// TIA Portal V17 export
// export: Created 2024-08-29T23:09:23.5181153Z, ExportSetting WithDefaults, DisplayName Totally Integrated Automation Portal, DisplayVersion V17 Update 7, DisplayName TIA Portal Openness, DisplayVersion V17 Update 7, DisplayName TIA Portal Version Control Interface, DisplayVersion V17, DisplayName SINAMICS Startdrive Advanced, DisplayVersion V17 SP2, DisplayName SINAMICS Startdrive G110M, G120, G120C, G120D, G120P, G115D, DisplayVersion V17 SP2, DisplayName SINAMICS Startdrive G130, G150, S120, S150, SINAMICS MV, S210, DisplayVersion V17 SP2, DisplayName STEP 7 Professional, DisplayVersion V17 Update 7, DisplayName STEP 7 Safety, DisplayVersion V17 Update 6, DisplayName WinCC Advanced / Unified PC, DisplayVersion V17 Update 7
FUNCTION "eksFC" : Void   // FC305, LAD
TITLE = Euchner Management EKS KEY
{ S7_Optimized_Access := 'FALSE' }
VERSION : 0.1
// stored: AutoNumber false, IsIECCheckEnabled false, SetENOAutomatically false, UDAEnableTagReadback false
   VAR_INPUT
      iKeyIn : Bool;
      iEksLevel : Byte;
      iEksEmployeeID : DWord;
      iEksKeyID1 : DWord;
      iEksKeyID2 : DWord;
      iEksJobFinished : Bool;
      hmiCurrentPage : Word;
   END_VAR
   VAR_OUTPUT
      qEksStartAdress : Byte;
      qEksDataLength : Byte;
      qEksData1 : Byte;
      qEksData2 : DWord;
      qEksWriteCommand : Bool;
   END_VAR
   VAR_TEMP
      tNone : Bool;
      tDBAddressKeys : Int;
      tDBAddressHMIPage : Int;
      tDBKeyStructLength : Int;
      tDBAddress : Int;
      tDBLength : Int;
      tCycle : Int;
      tFill : Int;
      tKey : "udt_EKS_KEY";
      tDBStartAddress : Int;
      tsearch : Bool;
      i : Int;
   END_VAR
   VAR CONSTANT
      DB : Byte := 16#84;
   END_VAR
   VAR_TEMP   // added for the SCL form of the ladder/FBD networks
      _w1 : Bool;
      _w2 : Bool;
   END_VAR
BEGIN

REGION Network 1: Initialize Temp Values
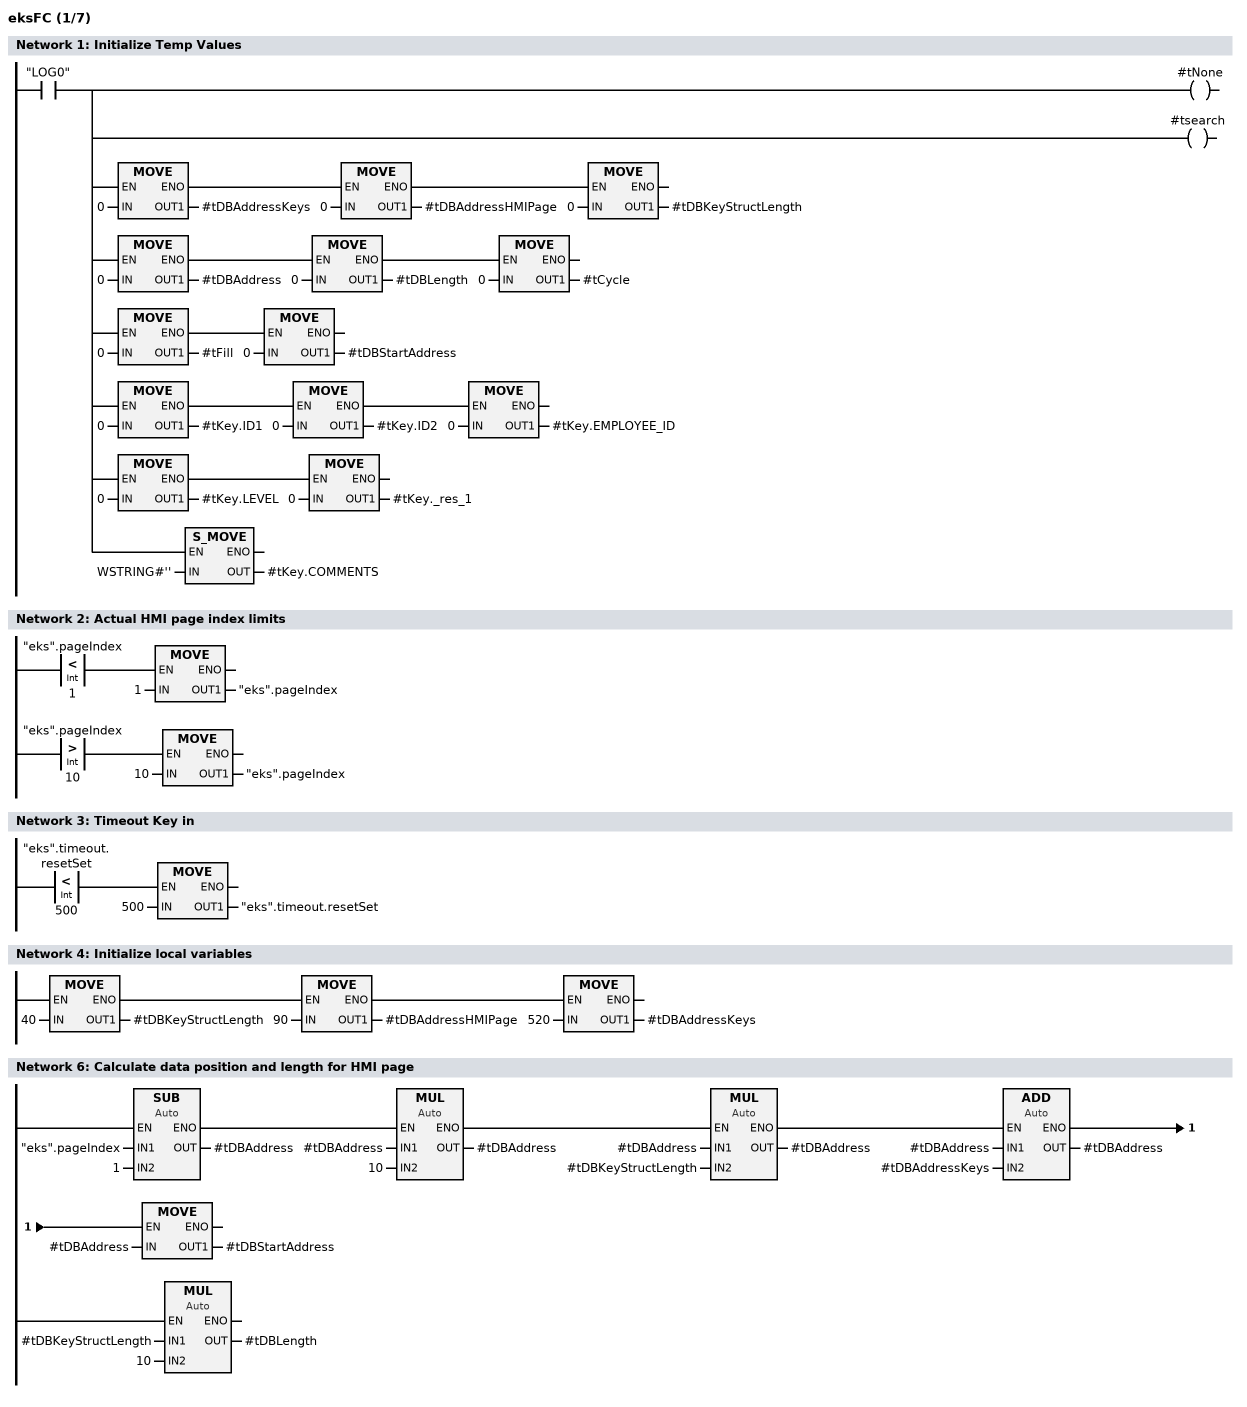
   RUNG wire#powerrail
      Contact( "LOG0" )
      wire#w1
      Coil( #tNone )
   END_RUNG
   RUNG wire#w1
      Coil( #tsearch )
   END_RUNG
   RUNG wire#w1
      Move(in := 0, out1 => #tDBAddressKeys)
      Move(in := 0, out1 => #tDBAddressHMIPage)
      Move(in := 0, out1 => #tDBKeyStructLength)
   END_RUNG
   RUNG wire#w1
      Move(in := 0, out1 => #tDBAddress)
      Move(in := 0, out1 => #tDBLength)
      Move(in := 0, out1 => #tCycle)
   END_RUNG
   RUNG wire#w1
      Move(in := 0, out1 => #tFill)
      Move(in := 0, out1 => #tDBStartAddress)
   END_RUNG
   RUNG wire#w1
      Move(in := 0, out1 => #tKey.ID1)
      Move(in := 0, out1 => #tKey.ID2)
      Move(in := 0, out1 => #tKey.EMPLOYEE_ID)
   END_RUNG
   RUNG wire#w1
      Move(in := 0, out1 => #tKey.LEVEL)
      Move(in := 0, out1 => #tKey._res_1)
   END_RUNG
   RUNG wire#w1
      S_Move(in := WSTRING#'', out => #tKey.COMMENTS)
   END_RUNG
   // the same network as SCL:
   #tNone := "LOG0";
   #tsearch := "LOG0";
   IF "LOG0" THEN
       #tDBAddressKeys := 0;
       #tDBAddressHMIPage := 0;
       #tDBKeyStructLength := 0;
       #tDBAddress := 0;
       #tDBLength := 0;
       #tCycle := 0;
       #tFill := 0;
       #tDBStartAddress := 0;
       #tKey.ID1 := 0;
       #tKey.ID2 := 0;
       #tKey.EMPLOYEE_ID := 0;
       #tKey.LEVEL := 0;
       #tKey._res_1 := 0;
       #tKey.COMMENTS := WSTRING#'';
   END_IF;
END_REGION

REGION Network 2: Actual HMI page index limits
   RUNG wire#powerrail
      { S7_Templates := "SrcType := Int" } LT_Contact(in1 := "eks".pageIndex, in2 := 1)
      Move(in := 1, out1 => "eks".pageIndex)
   END_RUNG
   RUNG wire#powerrail
      { S7_Templates := "SrcType := Int" } GT_Contact(in1 := "eks".pageIndex, in2 := 10)
      Move(in := 10, out1 => "eks".pageIndex)
   END_RUNG
   // the same network as SCL:
   IF "eks".pageIndex < 1 THEN "eks".pageIndex := 1; END_IF;
   IF "eks".pageIndex > 10 THEN "eks".pageIndex := 10; END_IF;
END_REGION

REGION Network 3: Timeout Key in
   RUNG wire#powerrail
      { S7_Templates := "SrcType := Int" } LT_Contact(in1 := "eks".timeout.resetSet, in2 := 500)
      Move(in := 500, out1 => "eks".timeout.resetSet)
   END_RUNG
   // the same network as SCL:
   IF "eks".timeout.resetSet < 500 THEN "eks".timeout.resetSet := 500; END_IF;
END_REGION

REGION Network 4: Initialize local variables
   RUNG wire#powerrail
      Move(in := 40, out1 => #tDBKeyStructLength)
      Move(in := 90, out1 => #tDBAddressHMIPage)
      Move(in := 520, out1 => #tDBAddressKeys)
   END_RUNG
   // the same network as SCL:
   #tDBKeyStructLength := 40;
   #tDBAddressHMIPage := 90;
   #tDBAddressKeys := 520;
END_REGION

REGION Network 6: Calculate data position and length for HMI page
   RUNG wire#powerrail
      Sub(in1 := "eks".pageIndex, in2 := 1, out => #tDBAddress)
      Mul(in1 := #tDBAddress, in2 := 10, out => #tDBAddress)
      Mul(in1 := #tDBAddress, in2 := #tDBKeyStructLength, out => #tDBAddress)
      Add(in1 := #tDBAddress, in2 := #tDBAddressKeys, out => #tDBAddress)
      Move(in := #tDBAddress, out1 => #tDBStartAddress)
   END_RUNG
   RUNG wire#powerrail
      Mul(in1 := #tDBKeyStructLength, in2 := 10, out => #tDBLength)
   END_RUNG
   // the same network as SCL:
   #tDBAddress := "eks".pageIndex - 1;
   #tDBAddress := #tDBAddress * 10;
   #tDBAddress := #tDBAddress * #tDBKeyStructLength;
   #tDBAddress := #tDBAddress + #tDBAddressKeys;
   #tDBStartAddress := #tDBAddress;
   #tDBLength := #tDBKeyStructLength * 10;
END_REGION

REGION Network 7 (SCL): Copy data for page (10 keys)
   POKE_BLK(area_src:=#DB,
            dbNumber_src:=305,
            byteOffset_src:=#tDBAddress,
            area_dest:=#DB,
            dbNumber_dest:=305,
            byteOffset_dest:=90,
            count:=#tDBLength);
END_REGION

REGION Network 9: Inserted key
   // Store_Key_In is used to display only 1 time the level of euchner during storage function.
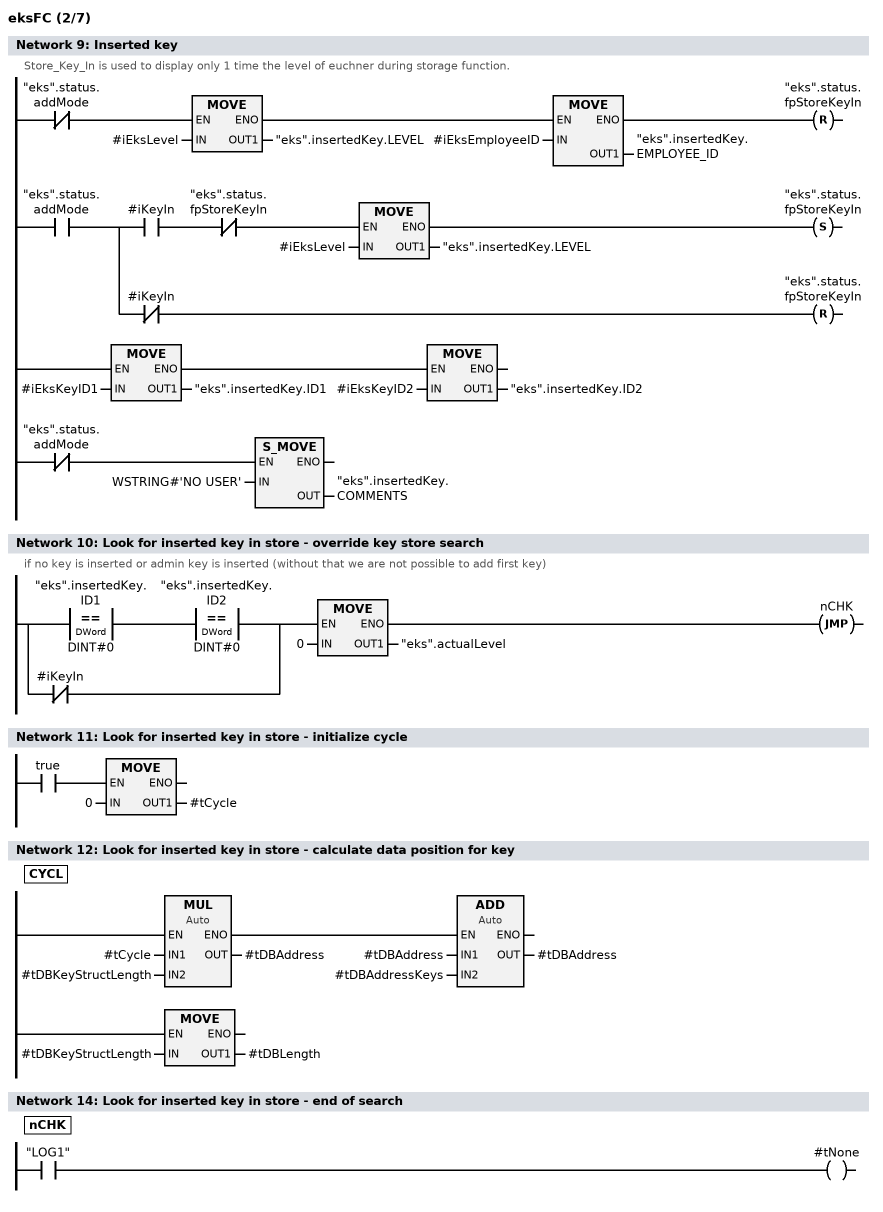
   RUNG wire#powerrail
      I_Contact( "eks".status.addMode )
      Move(in := #iEksLevel, out1 => "eks".insertedKey.LEVEL)
      Move(in := #iEksEmployeeID, out1 => "eks".insertedKey.EMPLOYEE_ID)
      R_Coil( "eks".status.fpStoreKeyIn )
   END_RUNG
   RUNG wire#powerrail
      Contact( "eks".status.addMode )
      wire#w1
      Contact( #iKeyIn )
      I_Contact( "eks".status.fpStoreKeyIn )
      Move(in := #iEksLevel, out1 => "eks".insertedKey.LEVEL)
      S_Coil( "eks".status.fpStoreKeyIn )
   END_RUNG
   RUNG wire#w1
      I_Contact( #iKeyIn )
      R_Coil( "eks".status.fpStoreKeyIn )
   END_RUNG
   RUNG wire#powerrail
      Move(in := #iEksKeyID1, out1 => "eks".insertedKey.ID1)
      Move(in := #iEksKeyID2, out1 => "eks".insertedKey.ID2)
   END_RUNG
   RUNG wire#powerrail
      I_Contact( "eks".status.addMode )
      S_Move(in := WSTRING#'NO USER', out => "eks".insertedKey.COMMENTS)
   END_RUNG
   // the same network as SCL:
   IF NOT "eks".status.addMode THEN
       "eks".insertedKey.LEVEL := #iEksLevel;
       "eks".insertedKey.EMPLOYEE_ID := #iEksEmployeeID;
       "eks".status.fpStoreKeyIn := FALSE;
   END_IF;
   IF "eks".status.addMode AND #iKeyIn AND NOT "eks".status.fpStoreKeyIn THEN
       "eks".insertedKey.LEVEL := #iEksLevel;
       "eks".status.fpStoreKeyIn := TRUE;
   END_IF;
   IF "eks".status.addMode AND NOT #iKeyIn THEN "eks".status.fpStoreKeyIn := FALSE; END_IF;
   "eks".insertedKey.ID1 := #iEksKeyID1;
   "eks".insertedKey.ID2 := #iEksKeyID2;
   IF NOT "eks".status.addMode THEN "eks".insertedKey.COMMENTS := WSTRING#'NO USER'; END_IF;
END_REGION

REGION Network 10: Look for inserted key in store - override key store search
   // if no key is inserted or admin key is inserted (without that we are not possible to add first key)
   RUNG wire#powerrail
      { S7_Templates := "SrcType := DWord" } EQ_Contact(in1 := "eks".insertedKey.ID1, in2 := DINT#0)
      { S7_Templates := "SrcType := DWord" } EQ_Contact(in1 := "eks".insertedKey.ID2, in2 := DINT#0)
      wire#w1
      Move(in := 0, out1 => "eks".actualLevel)
      JumpCoil( nCHK )
   END_RUNG
   RUNG wire#powerrail
      I_Contact( #iKeyIn )
   END_RUNG wire#w1
   // the same network as SCL:
   #_w1 := (("eks".insertedKey.ID1 = DINT#0) AND ("eks".insertedKey.ID2 = DINT#0)) OR NOT #iKeyIn;
   IF #_w1 THEN
       "eks".actualLevel := 0;
       GOTO nCHK;
   END_IF;
END_REGION

REGION Network 11: Look for inserted key in store - initialize cycle
   RUNG wire#powerrail
      Contact( true )
      Move(in := 0, out1 => #tCycle)
   END_RUNG
   // the same network as SCL:
   IF true THEN #tCycle := 0; END_IF;
END_REGION

REGION Network 12: Look for inserted key in store - calculate data position for key
   Label( CYCL )
   RUNG wire#powerrail
      Mul(in1 := #tCycle, in2 := #tDBKeyStructLength, out => #tDBAddress)
      Add(in1 := #tDBAddress, in2 := #tDBAddressKeys, out => #tDBAddress)
   END_RUNG
   RUNG wire#powerrail
      Move(in := #tDBKeyStructLength, out1 => #tDBLength)
   END_RUNG
   // the same network as SCL:
   CYCL:
   #tDBAddress := #tCycle * #tDBKeyStructLength;
   #tDBAddress := #tDBAddress + #tDBAddressKeys;
   #tDBLength := #tDBKeyStructLength;
END_REGION

REGION Network 13 (SCL): Look for inserted key in store - check ID of stored key
   FOR #i := 1 TO 130 DO
       #tKey := "eks".keys[#i];
       IF (#tKey.ID1 = "eks".insertedKey.ID1) AND
           (#tKey.ID2 = "eks".insertedKey.ID2) THEN
           "eks".actualLevel := #tKey.LEVEL;
           "eks".insertedKey.COMMENTS := #tKey.COMMENTS;
           EXIT;
       END_IF;
   END_FOR;
END_REGION

REGION Network 14: Look for inserted key in store - end of search
   Label( nCHK )
   RUNG wire#powerrail
      Contact( "LOG1" )
      Coil( #tNone )
   END_RUNG
   // the same network as SCL:
   nCHK:
   #tNone := "LOG1";
END_REGION

REGION Network 15: Reset of EKS higher levels until key is removed
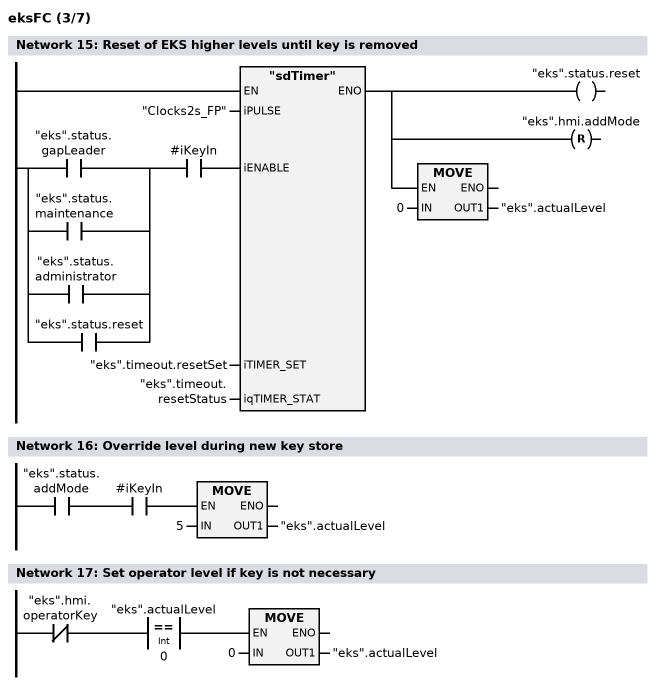
   RUNG wire#powerrail
      "sdTimer"(iENABLE := wire#w2, iPULSE := "Clocks2s_FP", iTIMER_SET := "eks".timeout.resetSet, iqTIMER_STAT := "eks".timeout.resetStatus)
      wire#w3
      Coil( "eks".status.reset )
   END_RUNG
   RUNG wire#powerrail
      Contact( "eks".status.gapLeader )
      wire#w1
      Contact( #iKeyIn )
   END_RUNG wire#w2
   RUNG wire#powerrail
      Contact( "eks".status.maintenance )
   END_RUNG wire#w1
   RUNG wire#powerrail
      Contact( "eks".status.administrator )
   END_RUNG wire#w1
   RUNG wire#powerrail
      Contact( "eks".status.reset )
   END_RUNG wire#w1
   RUNG wire#w3
      R_Coil( "eks".hmi.addMode )
   END_RUNG
   RUNG wire#w3
      Move(in := 0, out1 => "eks".actualLevel)
   END_RUNG
   // the same network as SCL:
   "sdTimer"(iPULSE := "Clocks2s_FP",
             iENABLE := ("eks".status.gapLeader OR "eks".status.maintenance OR "eks".status.administrator OR "eks".status.reset) AND #iKeyIn,
             iTIMER_SET := "eks".timeout.resetSet,
             iqTIMER_STAT := "eks".timeout.resetStatus,
             ENO => #_w1);
   "eks".status.reset := #_w1;
   IF #_w1 THEN
       "eks".hmi.addMode := FALSE;
       "eks".actualLevel := 0;
   END_IF;
END_REGION

REGION Network 16: Override level during new key store
   RUNG wire#powerrail
      Contact( "eks".status.addMode )
      Contact( #iKeyIn )
      Move(in := 5, out1 => "eks".actualLevel)
   END_RUNG
   // the same network as SCL:
   IF "eks".status.addMode AND #iKeyIn THEN "eks".actualLevel := 5; END_IF;
END_REGION

REGION Network 17: Set operator level if key is not necessary
   RUNG wire#powerrail
      I_Contact( "eks".hmi.operatorKey )
      { S7_Templates := "SrcType := Int" } EQ_Contact(in1 := "eks".actualLevel, in2 := 0)
      Move(in := 0, out1 => "eks".actualLevel)
   END_RUNG
   // the same network as SCL:
   IF NOT "eks".hmi.operatorKey AND ("eks".actualLevel = 0) THEN "eks".actualLevel := 0; END_IF;
END_REGION

REGION Network 18: EKS levels
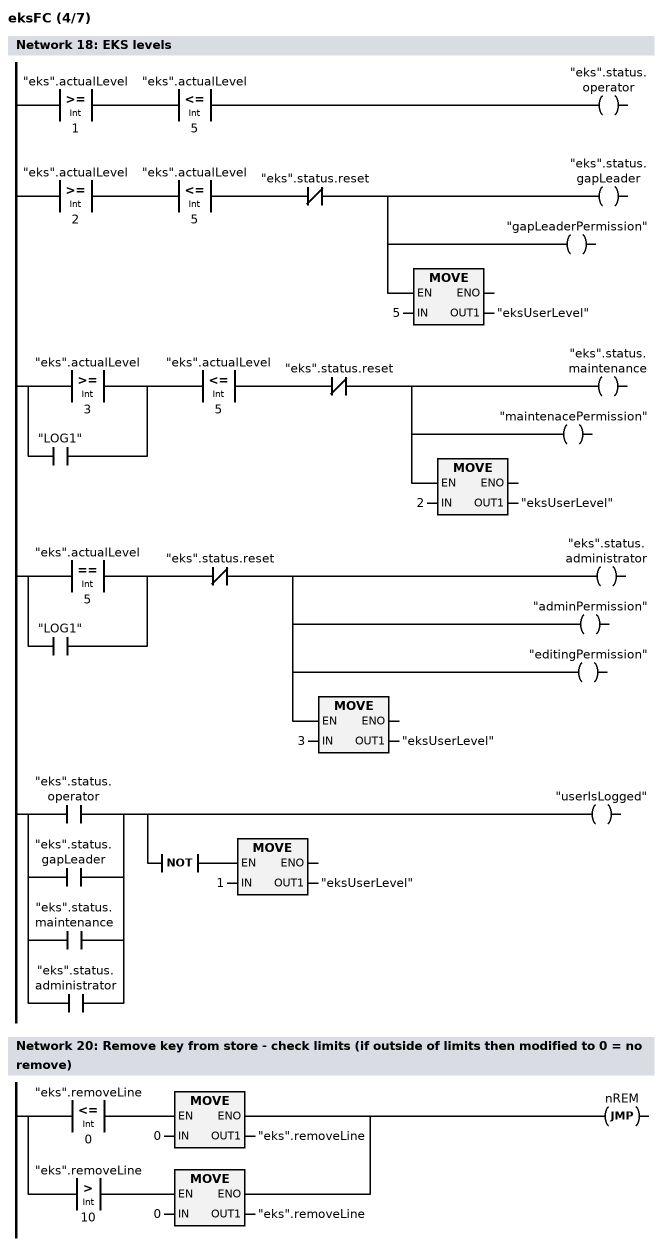
   RUNG wire#powerrail
      { S7_Templates := "SrcType := Int" } GE_Contact(in1 := "eks".actualLevel, in2 := 1)
      { S7_Templates := "SrcType := Int" } LE_Contact(in1 := "eks".actualLevel, in2 := 5)
      Coil( "eks".status.operator )
   END_RUNG
   RUNG wire#powerrail
      { S7_Templates := "SrcType := Int" } GE_Contact(in1 := "eks".actualLevel, in2 := 2)
      { S7_Templates := "SrcType := Int" } LE_Contact(in1 := "eks".actualLevel, in2 := 5)
      I_Contact( "eks".status.reset )
      wire#w1
      Coil( "eks".status.gapLeader )
   END_RUNG
   RUNG wire#w1
      Coil( "gapLeaderPermission" )
   END_RUNG
   RUNG wire#w1
      Move(in := 5, out1 => "eksUserLevel")
   END_RUNG
   RUNG wire#powerrail
      { S7_Templates := "SrcType := Int" } GE_Contact(in1 := "eks".actualLevel, in2 := 3)
      wire#w2
      { S7_Templates := "SrcType := Int" } LE_Contact(in1 := "eks".actualLevel, in2 := 5)
      I_Contact( "eks".status.reset )
      wire#w3
      Coil( "eks".status.maintenance )
   END_RUNG
   RUNG wire#powerrail
      Contact( "LOG1" )
   END_RUNG wire#w2
   RUNG wire#w3
      Coil( "maintenacePermission" )
   END_RUNG
   RUNG wire#w3
      Move(in := 2, out1 => "eksUserLevel")
   END_RUNG
   RUNG wire#powerrail
      { S7_Templates := "SrcType := Int" } EQ_Contact(in1 := "eks".actualLevel, in2 := 5)
      wire#w4
      I_Contact( "eks".status.reset )
      wire#w5
      Coil( "eks".status.administrator )
   END_RUNG
   RUNG wire#powerrail
      Contact( "LOG1" )
   END_RUNG wire#w4
   RUNG wire#w5
      Coil( "adminPermission" )
   END_RUNG
   RUNG wire#w5
      Coil( "editingPermission" )
   END_RUNG
   RUNG wire#w5
      Move(in := 3, out1 => "eksUserLevel")
   END_RUNG
   RUNG wire#powerrail
      Contact( "eks".status.operator )
      wire#w6
      Coil( "userIsLogged" )
   END_RUNG
   RUNG wire#powerrail
      Contact( "eks".status.gapLeader )
   END_RUNG wire#w6
   RUNG wire#powerrail
      Contact( "eks".status.maintenance )
   END_RUNG wire#w6
   RUNG wire#powerrail
      Contact( "eks".status.administrator )
   END_RUNG wire#w6
   RUNG wire#w6
      Not()
      Move(in := 1, out1 => "eksUserLevel")
   END_RUNG
   // the same network as SCL:
   "eks".status.operator := ("eks".actualLevel >= 1) AND ("eks".actualLevel <= 5);
   "eks".status.gapLeader := ("eks".actualLevel >= 2) AND ("eks".actualLevel <= 5) AND NOT "eks".status.reset;
   "gapLeaderPermission" := "eks".status.gapLeader;
   IF "eks".status.gapLeader THEN "eksUserLevel" := 5; END_IF;
   "eks".status.maintenance := (("eks".actualLevel >= 3) OR "LOG1") AND ("eks".actualLevel <= 5) AND NOT "eks".status.reset;
   "maintenacePermission" := "eks".status.maintenance;
   IF "eks".status.maintenance THEN "eksUserLevel" := 2; END_IF;
   "eks".status.administrator := (("eks".actualLevel = 5) OR "LOG1") AND NOT "eks".status.reset;
   "adminPermission" := "eks".status.administrator;
   "editingPermission" := "eks".status.administrator;
   IF "eks".status.administrator THEN "eksUserLevel" := 3; END_IF;
   "userIsLogged" := "eks".status.operator OR "eks".status.gapLeader OR "eks".status.maintenance OR "eks".status.administrator;
   IF NOT "userIsLogged" THEN "eksUserLevel" := 1; END_IF;
END_REGION

REGION Network 20: Remove key from store - check limits (if outside of limits then modified to 0 = no remove)
   RUNG wire#powerrail
      { S7_Templates := "SrcType := Int" } LE_Contact(in1 := "eks".removeLine, in2 := 0)
      Move(in := 0, out1 => "eks".removeLine)
      wire#w1
      JumpCoil( nREM )
   END_RUNG
   RUNG wire#powerrail
      { S7_Templates := "SrcType := Int" } GT_Contact(in1 := "eks".removeLine, in2 := 10)
      Move(in := 0, out1 => "eks".removeLine)
   END_RUNG wire#w1
   // the same network as SCL:
   #_w1 := "eks".removeLine <= 0;
   IF #_w1 THEN "eks".removeLine := 0; END_IF;
   #_w2 := "eks".removeLine > 10;
   IF #_w2 THEN "eks".removeLine := 0; END_IF;
   IF #_w1 OR #_w2 THEN GOTO nREM; END_IF;
END_REGION

REGION Network 21: Remove key from store - calculate data position and length for HMI page
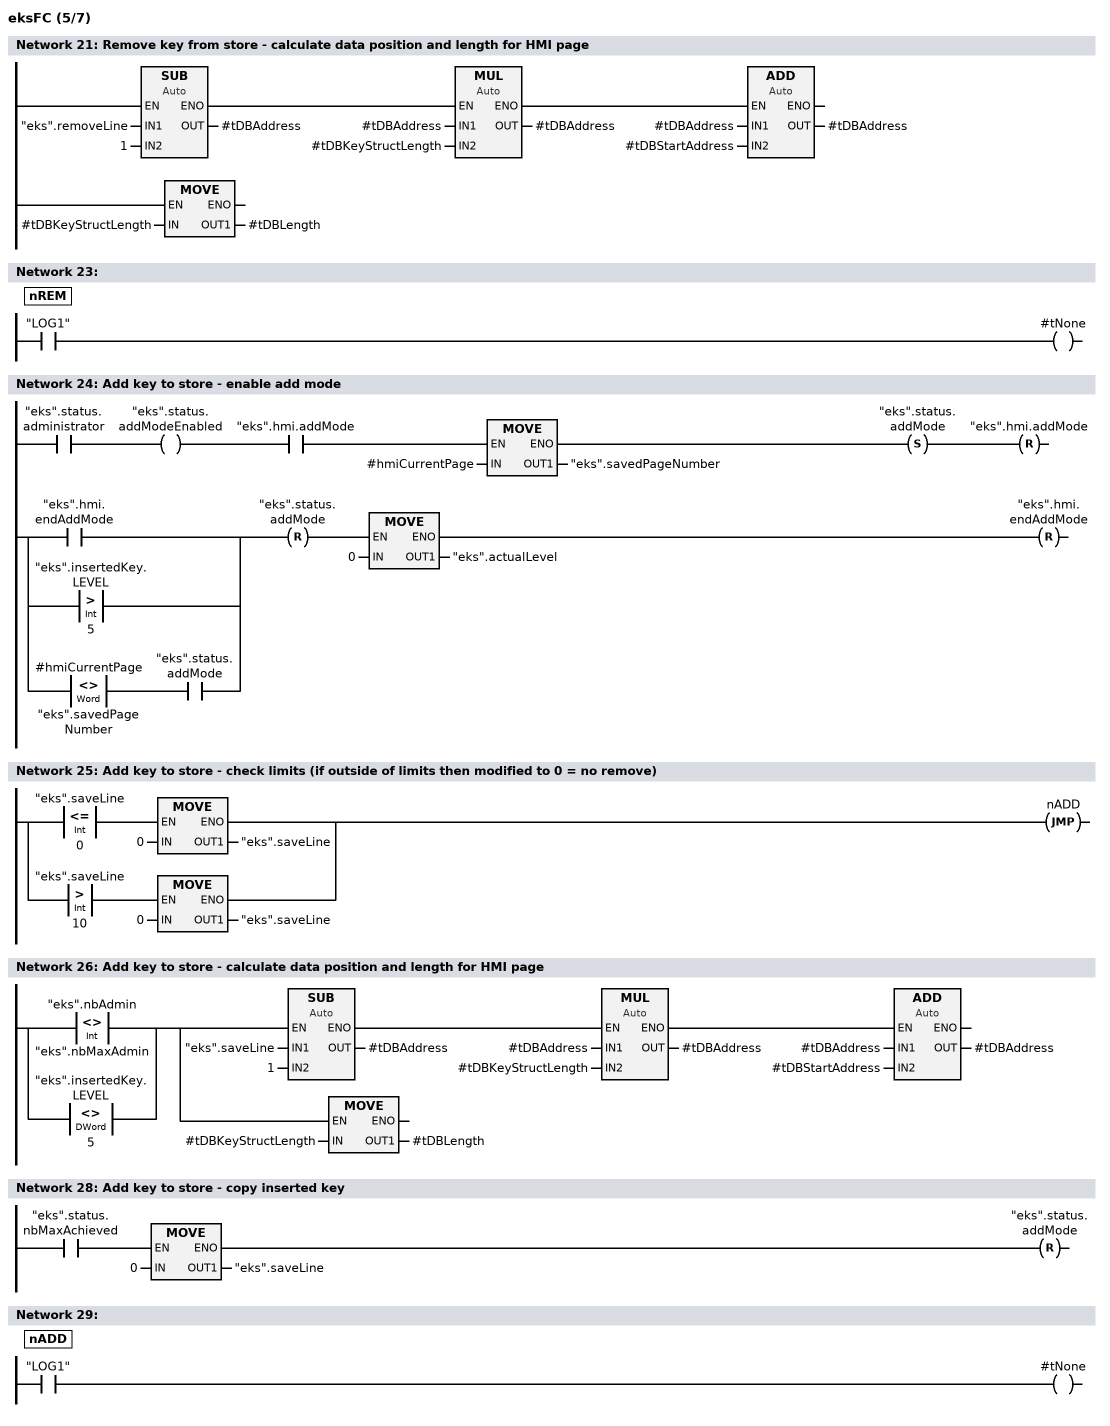
   RUNG wire#powerrail
      Sub(in1 := "eks".removeLine, in2 := 1, out => #tDBAddress)
      Mul(in1 := #tDBAddress, in2 := #tDBKeyStructLength, out => #tDBAddress)
      Add(in1 := #tDBAddress, in2 := #tDBStartAddress, out => #tDBAddress)
   END_RUNG
   RUNG wire#powerrail
      Move(in := #tDBKeyStructLength, out1 => #tDBLength)
   END_RUNG
   // the same network as SCL:
   #tDBAddress := "eks".removeLine - 1;
   #tDBAddress := #tDBAddress * #tDBKeyStructLength;
   #tDBAddress := #tDBAddress + #tDBStartAddress;
   #tDBLength := #tDBKeyStructLength;
END_REGION

REGION Network 22 (SCL): Remove key from store - delete key
   #tFill := 0;

   POKE_BLK(area_src:=#DB,
            dbNumber_src:=305,
            byteOffset_src:=5720,
            area_dest:=#DB,
            dbNumber_dest:=305,
            byteOffset_dest:=#tDBAddress,
            count:=#tDBLength);

   "eks".removeLine := 0;
END_REGION

REGION Network 23
   Label( nREM )
   RUNG wire#powerrail
      Contact( "LOG1" )
      Coil( #tNone )
   END_RUNG
   // the same network as SCL:
   nREM:
   #tNone := "LOG1";
END_REGION

REGION Network 24: Add key to store - enable add mode
   RUNG wire#powerrail
      Contact( "eks".status.administrator )
      Coil( "eks".status.addModeEnabled )
      Contact( "eks".hmi.addMode )
      Move(in := #hmiCurrentPage, out1 => "eks".savedPageNumber)
      S_Coil( "eks".status.addMode )
      R_Coil( "eks".hmi.addMode )
   END_RUNG
   RUNG wire#powerrail
      Contact( "eks".hmi.endAddMode )
      wire#w1
      R_Coil( "eks".status.addMode )
      Move(in := 0, out1 => "eks".actualLevel)
      R_Coil( "eks".hmi.endAddMode )
   END_RUNG
   RUNG wire#powerrail
      { S7_Templates := "SrcType := Int" } GT_Contact(in1 := "eks".insertedKey.LEVEL, in2 := 5)
   END_RUNG wire#w1
   RUNG wire#powerrail
      { S7_Templates := "SrcType := Word" } NE_Contact(in1 := #hmiCurrentPage, in2 := "eks".savedPageNumber)
      Contact( "eks".status.addMode )
   END_RUNG wire#w1
   // the same network as SCL:
   "eks".status.addModeEnabled := "eks".status.administrator;
   IF "eks".status.administrator AND "eks".hmi.addMode THEN
       "eks".savedPageNumber := #hmiCurrentPage;
       "eks".status.addMode := TRUE;
       "eks".hmi.addMode := FALSE;
   END_IF;
   #_w1 := "eks".hmi.endAddMode OR ("eks".insertedKey.LEVEL > 5) OR ((#hmiCurrentPage <> "eks".savedPageNumber) AND "eks".status.addMode);
   IF #_w1 THEN
       "eks".status.addMode := FALSE;
       "eks".actualLevel := 0;
       "eks".hmi.endAddMode := FALSE;
   END_IF;
END_REGION

REGION Network 25: Add key to store - check limits (if outside of limits then modified to 0 = no remove)
   RUNG wire#powerrail
      { S7_Templates := "SrcType := Int" } LE_Contact(in1 := "eks".saveLine, in2 := 0)
      Move(in := 0, out1 => "eks".saveLine)
      wire#w1
      JumpCoil( nADD )
   END_RUNG
   RUNG wire#powerrail
      { S7_Templates := "SrcType := Int" } GT_Contact(in1 := "eks".saveLine, in2 := 10)
      Move(in := 0, out1 => "eks".saveLine)
   END_RUNG wire#w1
   // the same network as SCL:
   #_w1 := "eks".saveLine <= 0;
   IF #_w1 THEN "eks".saveLine := 0; END_IF;
   #_w2 := "eks".saveLine > 10;
   IF #_w2 THEN "eks".saveLine := 0; END_IF;
   IF #_w1 OR #_w2 THEN GOTO nADD; END_IF;
END_REGION

REGION Network 26: Add key to store - calculate data position and length for HMI page
   RUNG wire#powerrail
      { S7_Templates := "SrcType := Int" } NE_Contact(in1 := "eks".nbAdmin, in2 := "eks".nbMaxAdmin)
      wire#w1
      Sub(in1 := "eks".saveLine, in2 := 1, out => #tDBAddress)
      Mul(in1 := #tDBAddress, in2 := #tDBKeyStructLength, out => #tDBAddress)
      Add(in1 := #tDBAddress, in2 := #tDBStartAddress, out => #tDBAddress)
   END_RUNG
   RUNG wire#powerrail
      { S7_Templates := "SrcType := DWord" } NE_Contact(in1 := "eks".insertedKey.LEVEL, in2 := 5)
   END_RUNG wire#w1
   RUNG wire#w1
      Move(in := #tDBKeyStructLength, out1 => #tDBLength)
   END_RUNG
   // the same network as SCL:
   IF ("eks".nbAdmin <> "eks".nbMaxAdmin) OR ("eks".insertedKey.LEVEL <> 5) THEN
       #tDBAddress := "eks".saveLine - 1;
       #tDBAddress := #tDBAddress * #tDBKeyStructLength;
       #tDBAddress := #tDBAddress + #tDBStartAddress;
       #tDBLength := #tDBKeyStructLength;
   END_IF;
END_REGION

REGION Network 27 (SCL): Add key to store - copy inserted key
   IF ("eks".insertedKey.LEVEL = 5  & NOT "eks".status.nbMaxAchieved) OR
       ("eks".insertedKey.LEVEL <> 5) THEN
       POKE_BLK(area_src := #DB,
                dbNumber_src := 305,
                byteOffset_src := 50,
                area_dest := #DB,
                dbNumber_dest := 305,
                byteOffset_dest := #tDBAddress,
                count := #tDBLength);
      "eks".saveLine := 0;
   END_IF;
END_REGION

REGION Network 28: Add key to store - copy inserted key
   RUNG wire#powerrail
      Contact( "eks".status.nbMaxAchieved )
      Move(in := 0, out1 => "eks".saveLine)
      R_Coil( "eks".status.addMode )
   END_RUNG
   // the same network as SCL:
   IF "eks".status.nbMaxAchieved THEN
       "eks".saveLine := 0;
       "eks".status.addMode := FALSE;
   END_IF;
END_REGION

REGION Network 29
   Label( nADD )
   RUNG wire#powerrail
      Contact( "LOG1" )
      Coil( #tNone )
   END_RUNG
   // the same network as SCL:
   nADD:
   #tNone := "LOG1";
END_REGION

REGION Network 30
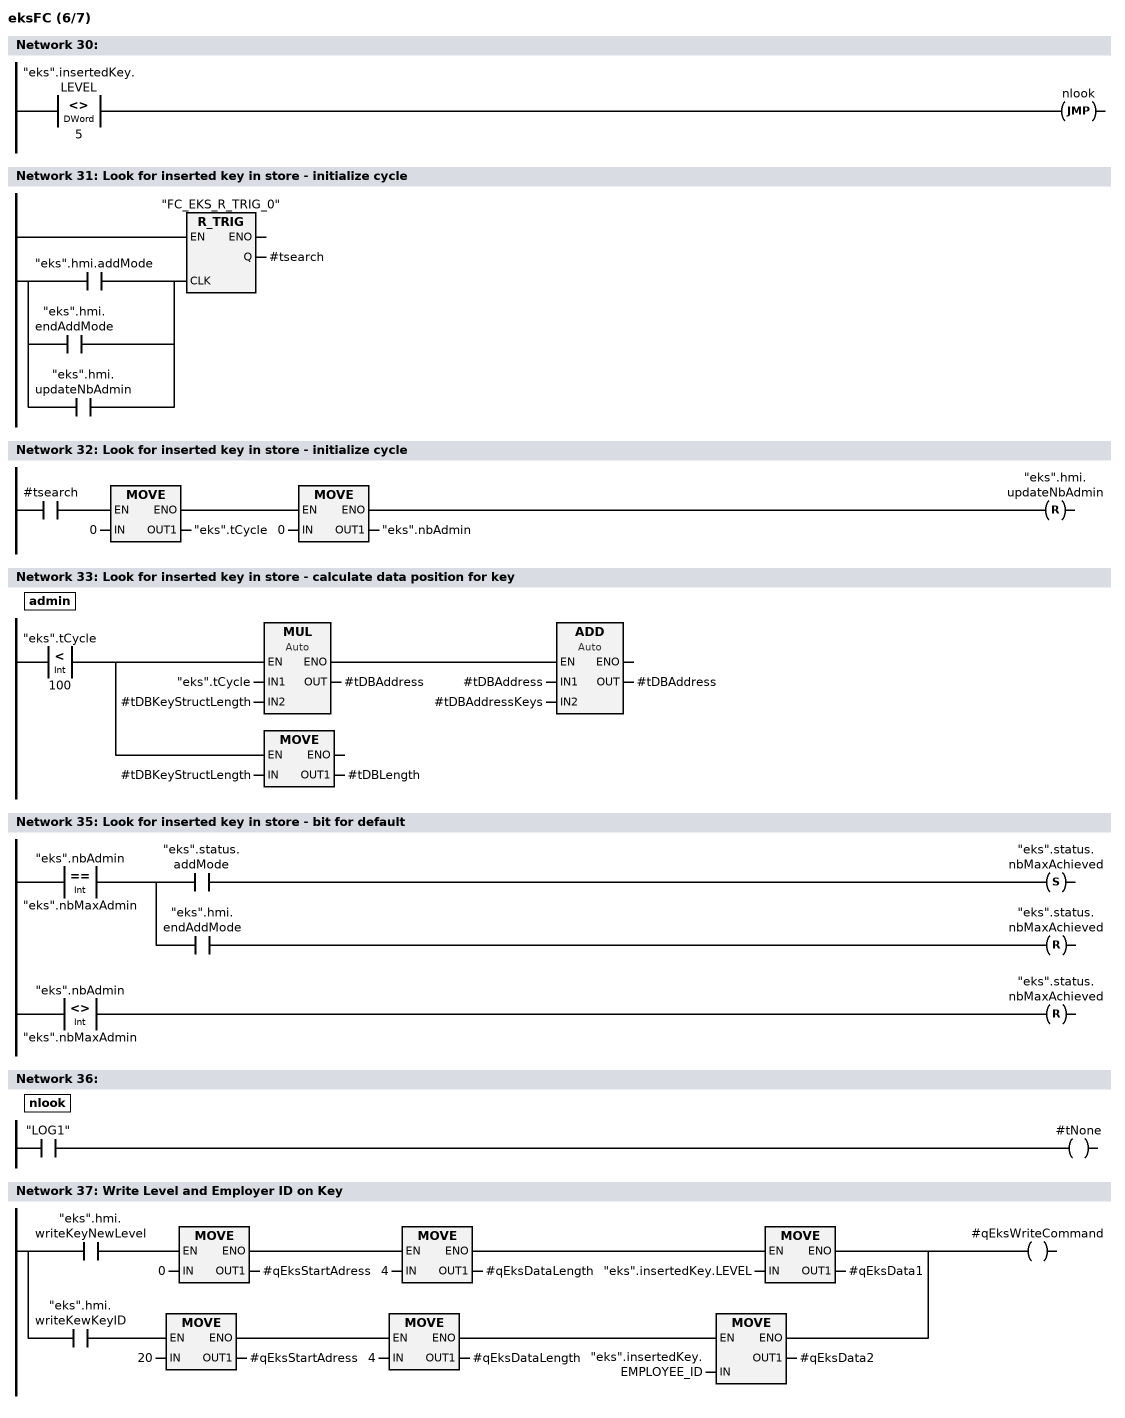
   RUNG wire#powerrail
      { S7_Templates := "SrcType := DWord" } NE_Contact(in1 := "eks".insertedKey.LEVEL, in2 := 5)
      JumpCoil( nlook )
   END_RUNG
   // the same network as SCL:
   IF "eks".insertedKey.LEVEL <> 5 THEN GOTO nlook; END_IF;
END_REGION

REGION Network 31: Look for inserted key in store - initialize cycle
   RUNG wire#powerrail
      "FC_EKS_R_TRIG_0".R_TRIG(CLK := wire#w1, Q => #tsearch)
   END_RUNG
   RUNG wire#powerrail
      Contact( "eks".hmi.addMode )
   END_RUNG wire#w1
   RUNG wire#powerrail
      Contact( "eks".hmi.endAddMode )
   END_RUNG wire#w1
   RUNG wire#powerrail
      Contact( "eks".hmi.updateNbAdmin )
   END_RUNG wire#w1
   // the same network as SCL:
   "FC_EKS_R_TRIG_0"(CLK := "eks".hmi.addMode OR "eks".hmi.endAddMode OR "eks".hmi.updateNbAdmin, Q => #tsearch);   // R_TRIG
END_REGION

REGION Network 32: Look for inserted key in store - initialize cycle
   RUNG wire#powerrail
      Contact( #tsearch )
      Move(in := 0, out1 => "eks".tCycle)
      Move(in := 0, out1 => "eks".nbAdmin)
      R_Coil( "eks".hmi.updateNbAdmin )
   END_RUNG
   // the same network as SCL:
   IF #tsearch THEN
       "eks".tCycle := 0;
       "eks".nbAdmin := 0;
       "eks".hmi.updateNbAdmin := FALSE;
   END_IF;
END_REGION

REGION Network 33: Look for inserted key in store - calculate data position for key
   Label( admin )
   RUNG wire#powerrail
      { S7_Templates := "SrcType := Int" } LT_Contact(in1 := "eks".tCycle, in2 := 100)
      wire#w1
      Mul(in1 := "eks".tCycle, in2 := #tDBKeyStructLength, out => #tDBAddress)
      Add(in1 := #tDBAddress, in2 := #tDBAddressKeys, out => #tDBAddress)
   END_RUNG
   RUNG wire#w1
      Move(in := #tDBKeyStructLength, out1 => #tDBLength)
   END_RUNG
   // the same network as SCL:
   admin:
   IF "eks".tCycle < 100 THEN
       #tDBAddress := "eks".tCycle * #tDBKeyStructLength;
       #tDBAddress := #tDBAddress + #tDBAddressKeys;
       #tDBLength := #tDBKeyStructLength;
   END_IF;
END_REGION

REGION Network 34 (SCL): Look for inserted key in store - check ID of stored key
   FOR #i := 1 TO 100 DO
       #tKey := "eks".keys[#i];
       IF #tKey.LEVEL = 5 THEN
           "eks".nbAdmin += 1;
           CONTINUE;
       END_IF;
   END_FOR;
END_REGION

REGION Network 35: Look for inserted key in store - bit for default
   RUNG wire#powerrail
      { S7_Templates := "SrcType := Int" } EQ_Contact(in1 := "eks".nbAdmin, in2 := "eks".nbMaxAdmin)
      wire#w1
      Contact( "eks".status.addMode )
      S_Coil( "eks".status.nbMaxAchieved )
   END_RUNG
   RUNG wire#w1
      Contact( "eks".hmi.endAddMode )
      R_Coil( "eks".status.nbMaxAchieved )
   END_RUNG
   RUNG wire#powerrail
      { S7_Templates := "SrcType := Int" } NE_Contact(in1 := "eks".nbAdmin, in2 := "eks".nbMaxAdmin)
      R_Coil( "eks".status.nbMaxAchieved )
   END_RUNG
   // the same network as SCL:
   #_w1 := "eks".nbAdmin = "eks".nbMaxAdmin;
   IF #_w1 AND "eks".status.addMode THEN "eks".status.nbMaxAchieved := TRUE; END_IF;
   IF #_w1 AND "eks".hmi.endAddMode THEN "eks".status.nbMaxAchieved := FALSE; END_IF;
   IF "eks".nbAdmin <> "eks".nbMaxAdmin THEN "eks".status.nbMaxAchieved := FALSE; END_IF;
END_REGION

REGION Network 36
   Label( nlook )
   RUNG wire#powerrail
      Contact( "LOG1" )
      Coil( #tNone )
   END_RUNG
   // the same network as SCL:
   nlook:
   #tNone := "LOG1";
END_REGION

REGION Network 37: Write Level and Employer ID on Key
   RUNG wire#powerrail
      Contact( "eks".hmi.writeKeyNewLevel )
      Move(in := 0, out1 => #qEksStartAdress)
      Move(in := 4, out1 => #qEksDataLength)
      Move(in := "eks".insertedKey.LEVEL, out1 => #qEksData1)
      wire#w1
      Coil( #qEksWriteCommand )
   END_RUNG
   RUNG wire#powerrail
      Contact( "eks".hmi.writeKewKeyID )
      Move(in := 20, out1 => #qEksStartAdress)
      Move(in := 4, out1 => #qEksDataLength)
      Move(in := "eks".insertedKey.EMPLOYEE_ID, out1 => #qEksData2)
   END_RUNG wire#w1
   // the same network as SCL:
   IF "eks".hmi.writeKeyNewLevel THEN
       #qEksStartAdress := 0;
       #qEksDataLength := 4;
       #qEksData1 := "eks".insertedKey.LEVEL;
   END_IF;
   IF "eks".hmi.writeKewKeyID THEN
       #qEksStartAdress := 20;
       #qEksDataLength := 4;
       #qEksData2 := "eks".insertedKey.EMPLOYEE_ID;
   END_IF;
   #qEksWriteCommand := "eks".hmi.writeKeyNewLevel OR "eks".hmi.writeKewKeyID;
END_REGION

REGION Network 38: Write Level and Employer ID on Key
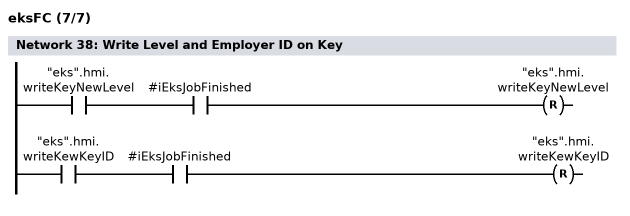
   RUNG wire#powerrail
      Contact( "eks".hmi.writeKeyNewLevel )
      Contact( #iEksJobFinished )
      R_Coil( "eks".hmi.writeKeyNewLevel )
   END_RUNG
   RUNG wire#powerrail
      Contact( "eks".hmi.writeKewKeyID )
      Contact( #iEksJobFinished )
      R_Coil( "eks".hmi.writeKewKeyID )
   END_RUNG
   // the same network as SCL:
   IF "eks".hmi.writeKeyNewLevel AND #iEksJobFinished THEN "eks".hmi.writeKeyNewLevel := FALSE; END_IF;
   IF "eks".hmi.writeKewKeyID AND #iEksJobFinished THEN "eks".hmi.writeKewKeyID := FALSE; END_IF;
END_REGION
END_FUNCTION
